REGION Network 31: Mapping of the process output data, control word 1, Bit 13
   #PO.x_Bit_13_Activate_Output_Stage_Inhibit := #ACTIVATE_OUTPUT_STAGE_INHIBIT;
END_REGION

REGION Network 32: Mapping of the process output data, control word 1, Bit 14
   #PO.x_Bit_14_Activate_StandBy_Mode := #ACTIVATE_STANDBY;
END_REGION

REGION Network 33: Mapping of the process output data, control word 1, Bit 15
   #PO.x_Bit_15_Heartbeat_IN := #HEARBEAT_IN;
END_REGION

REGION Network 34: Set the not used Bits to "false"
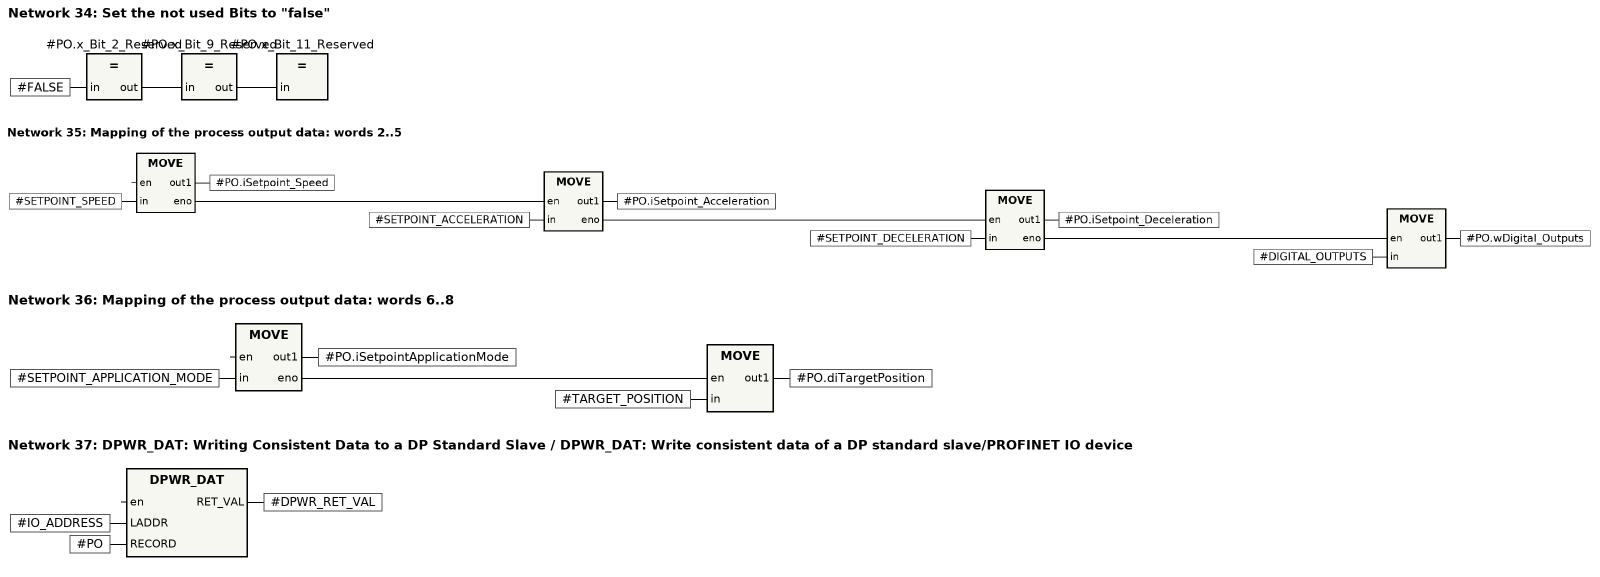
   #PO.x_Bit_2_Reserved := #FALSE;
   #PO.x_Bit_9_Reserved := #FALSE;
   #PO.x_Bit_11_Reserved := #FALSE;
END_REGION

REGION Network 35: Mapping of the process output data: words 2..5
   // ENO of a box is taken as its EN; it also drops when the box reports an error
   #PO.iSetpoint_Speed := #SETPOINT_SPEED;
   #PO.iSetpoint_Acceleration := #SETPOINT_ACCELERATION;
   #PO.iSetpoint_Deceleration := #SETPOINT_DECELERATION;
   #PO.wDigital_Outputs := #DIGITAL_OUTPUTS;
END_REGION

REGION Network 36: Mapping of the process output data: words 6..8
   // ENO of a box is taken as its EN; it also drops when the box reports an error
   #PO.iSetpointApplicationMode := #SETPOINT_APPLICATION_MODE;
   #PO.diTargetPosition := #TARGET_POSITION;
END_REGION

REGION Network 37: DPWR_DAT: Writing Consistent Data to a DP Standard Slave / DPWR_DAT: Write consistent data of a DP standard slave/PROFINET IO device
   // If the DPWR_DAT is processed without errors, the process output data is written consistently. If RET_VAL <> is 0, then there is an error.
   #DPWR_RET_VAL := DPWR_DAT(LADDR := #IO_ADDRESS, RECORD := #PO);
END_REGION

REGION Network 38: Erase FC outputs in case of an error (DPRD/WR_RET_VAL <> 0) / If processing of SFCs is faulty, all outputs of function will be deleted
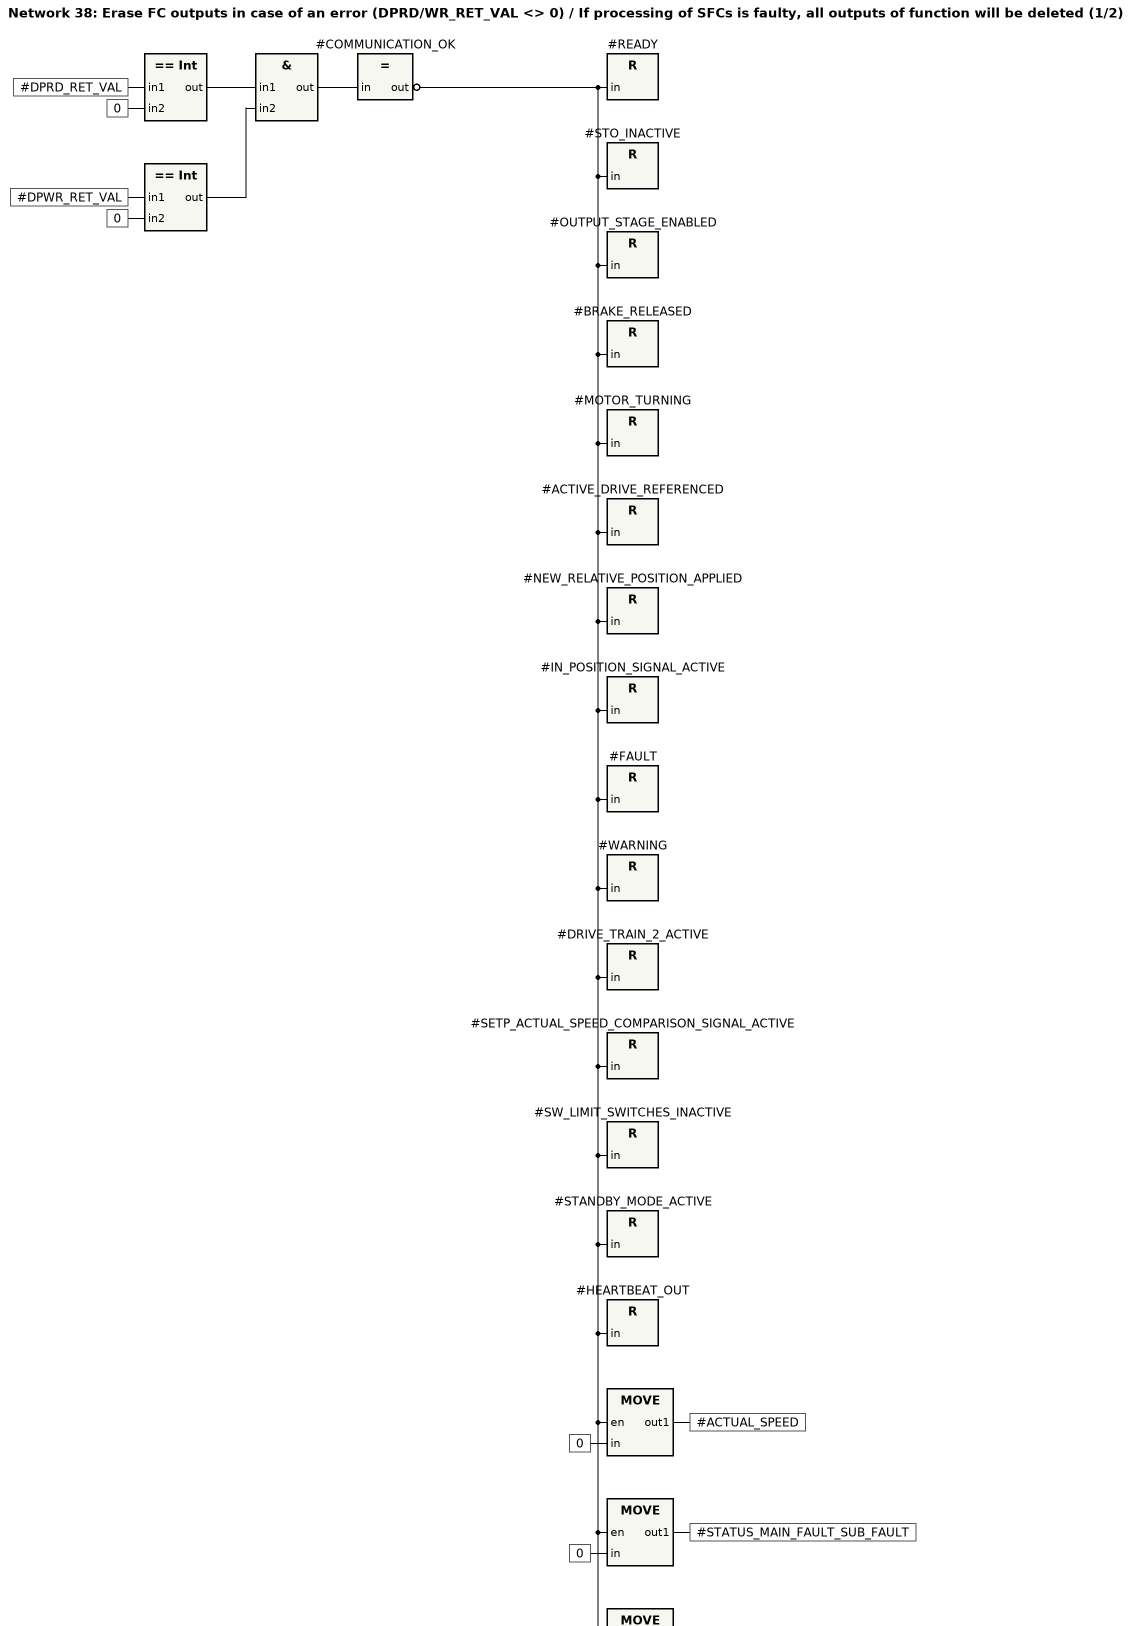
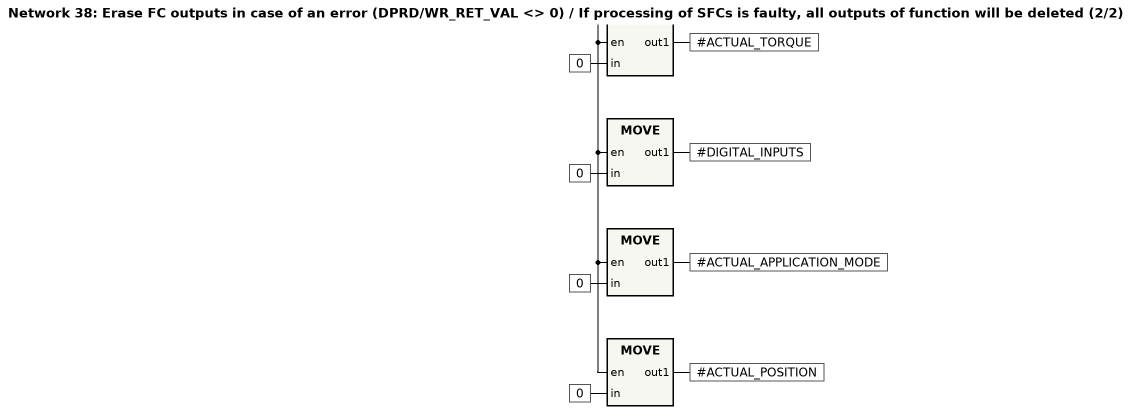
   END:
   #_w1 := (#DPRD_RET_VAL = 0) AND (#DPWR_RET_VAL = 0);
   #COMMUNICATION_OK := #_w1;
   IF NOT #_w1 THEN
       #READY := FALSE;
       #STO_INACTIVE := FALSE;
       #OUTPUT_STAGE_ENABLED := FALSE;
       #BRAKE_RELEASED := FALSE;
       #MOTOR_TURNING := FALSE;
       #ACTIVE_DRIVE_REFERENCED := FALSE;
       #NEW_RELATIVE_POSITION_APPLIED := FALSE;
       #IN_POSITION_SIGNAL_ACTIVE := FALSE;
       #FAULT := FALSE;
       #WARNING := FALSE;
       #DRIVE_TRAIN_2_ACTIVE := FALSE;
       #SETP_ACTUAL_SPEED_COMPARISON_SIGNAL_ACTIVE := FALSE;
       #SW_LIMIT_SWITCHES_INACTIVE := FALSE;
       #STANDBY_MODE_ACTIVE := FALSE;
       #HEARTBEAT_OUT := FALSE;
       #ACTUAL_SPEED := 0;
       #STATUS_MAIN_FAULT_SUB_FAULT := 0;
       #ACTUAL_TORQUE := 0;
       #DIGITAL_INPUTS := 0;
       #ACTUAL_APPLICATION_MODE := 0;
       #ACTUAL_POSITION := 0;
   END_IF;
END_REGION
END_FUNCTION

ORGANIZATION_BLOCK "Main"   // OB1, FBD
TITLE = "Main Program Sweep (Cycle)"
{ S7_Optimized_Access := 'FALSE' }
VERSION : 0.1
// This sample program only demonstrates the basic approach. We do not accept any legal or other liability for incorrect program functions and their consequences!
   VAR_TEMP
      OB1_EV_CLASS : Byte;   // Bits 0-3 = 1 (Coming event), Bits 4-7 = 1 (Event class 1)
      OB1_SCAN_1 : Byte;   // 1 (Cold restart scan 1 of OB 1), 3 (Scan 2-n of OB 1)
      OB1_PRIORITY : Byte;   // Priority of OB Execution
      OB1_OB_NUMBR : Byte;   // 1 (Organization block 1, OB1)
      OB1_RESERVED_1 : Byte;   // Reserved for system
      OB1_RESERVED_2 : Byte;   // Reserved for system
      OB1_PREV_CYCLE : Int;   // Cycle time of previous OB1 scan (milliseconds)
      OB1_MIN_CYCLE : Int;   // Minimum cycle time of OB1 (milliseconds)
      OB1_MAX_CYCLE : Int;   // Maximum cycle time of OB1 (milliseconds)
      OB1_DATE_TIME : Date_And_Time;   // Date and time OB1 started
   END_VAR
BEGIN

REGION Network 1: Control of the drive pos-UDT-s73xx
   // Please take note of the manual "MOVIKIT® Positioning, Velocity"
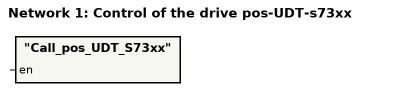
   "Call_pos_UDT_S73xx"();
END_REGION
END_ORGANIZATION_BLOCK